Staubli VAL3: IPMove.pgx

public program IPMove()
begin
  //
//  $XgetDrvCmdPos(nDrvPos)
//  for l_i=0 to nAxesSum-1
//    aioSet(aoIPPos[l_i],(nDrvPos[l_i]*nResolution[l_i]/nScaleFact[l_i]))
//  endFor
end
